{attribute addProperty BoxType "EP2328-1061-0016"}
{attribute addProperty Id "InputAT %I*BOOL81"}
{attribute addProperty CRC "3836671390"}
{attribute addProperty SizeInBites "8"}
{attribute addProperty SizeInBytes "1"}
TYPE DI_X01_Pin2_Input_E4AEF59E :
STRUCT
	{attribute addProperty Name "Input"}
	Input AT %I* : BOOL;
END_STRUCT
END_TYPE

(* stored: Version 1.2.0.0, ProductVersion 3.1.4024.9
   DUT DI_X01_Pin2_Input_E4AEF59E: Id {564f09a1-3cce-417a-ba18-06ac358535d9} *)
